# EPICS IOC start-up script: tcs-mk-iocApp/config/tcs.subs
dbLoadRecords ("db/tcsTop.db","top=tcs:,tcs=tcs:,m2=m2:,ag=ag:,mc=mc:,cr=cr:,ao=ao:,m1=m1:,ec=ec:,ws=ws:,gp=tcs:gp:,sad=tcs:sad:,pwfs1=pwfs1:,pwfs2=pwfs2:,hrwfs=hrwfs:,oiwfs=oiwfs:,nici=tcs:nici:,aom=tcs:aom:,gsaoi=tgsaoi:,gems=tcs:gems:")

dbLoadRecords ("db/tcsSad.db","top=tcs:,tcs=tcs:,sad=tcs:sad:")

dbLoadRecords ("db/tcsSimulations.db","top=tcs:,tcs=tcs:,m2=tcs:m2:,ag=tcs:ag:,mc=tcs:mc:,cr=tcs:cr:,ao=tcs:ao:,m1=tcs:m1:,ec=tcs:ec:,ws=tcs:ws:,gp=tcs:gp:,pwfs1=tpwfs1:,pwfs2=tpwfs2:,oiwfs=toiwfs:,nici=tcs:nici:,aom=tcs:aom:,gsaoi=tgsaoi:,gems=tcs:gems:,gi=tcs:gi:")
